# EPICS autosave request: sscan/sscanApp/Db/standardScans_settings.req
file sscanRecord_settings.req P=$(P),S=scan1
file sscanRecord_settings.req P=$(P),S=scan2
file sscanRecord_settings.req P=$(P),S=scan3
file sscanRecord_settings.req P=$(P),S=scan4
file sscanRecord_settings.req P=$(P),S=scanH
